% RSLogix 500 project One Button OSR.RSS, saved by version 10.00.00.00 %
PROJECT "MWL"    % processor: Bul.1763 MicroLogix 1100 Series B %

PROGRAM FILES
  LAD 2   3 rungs

DATA FILES
  O0 OUTPUT  4 elements
  I1 INPUT  6 elements
  S2 STATUS  66 elements
  B3 BINARY  2 elements
  T4 TIMER  1 elements
  C5 COUNTER  1 elements
  R6 CONTROL  1 elements
  N7 INTEGER  1 elements
  F8 FLOAT  1 elements

LADDER 2
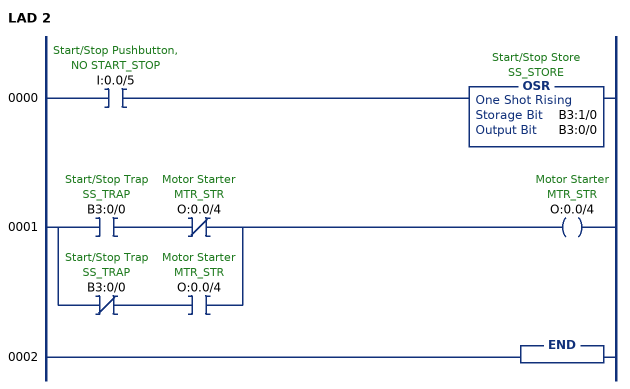
% Rung: 0 %
SOR XIC I:0.0/5 OSR B3:1/0 B3:0/0 EOR
%   I:0.0/5  START_STOP  "Start/Stop Pushbutton, NO" %
%   B3:1/0  SS_STORE  "Start/Stop Store" %
%   B3:0/0  SS_TRAP  "Start/Stop Trap" %
% Rung: 1 %
SOR BST XIC B3:0/0 XIO O:0.0/4 NXB XIO B3:0/0 XIC O:0.0/4 BND OTE O:0.0/4 EOR
%   B3:0/0  SS_TRAP  "Start/Stop Trap" %
%   O:0.0/4  MTR_STR  "Motor Starter" %
% Rung: 2 %
SOR END EOR
